# B&R Automation Studio project A2019059_Linka_Power_CP (part 14)

#### ProfinetKomunikaciaCU.st
```iecst
ACTION ProfinetKomunikaciaCU:

	//Stavy jednotky pre ovládanie kamier//
	ControlUnit.Stav_READY:= ControlUnit.Profinet_PLC_INPUTS[0].0;

END_ACTION
```

### Program Logical/Program/Linka/OvladanieSafety (IEC)

#### Main.st - Init, cyclic, exit code
```iecst
PROGRAM _INIT
	(* Insert code here *)

END_PROGRAM

PROGRAM _CYCLIC

	//*************************************Príznak tlačítka CS odblokované**********************************************//
	IF Safety.STAV.P1_Panel_TlacitkoCS_AKTIVNE AND
		Safety.STAV.P1_Robot_TlacitkoCS_AKTIVNE AND
		Safety.STAV.P1_Skrina_TlacitkoCS_AKTIVNE AND
		Safety.STAV.P2_Panel_TlacitkoCS_AKTIVNE AND
		Safety.STAV.P2_TlacitkoCS_AKTIVNE AND
		Safety.STAV.P2_Robot_TlacitkoCS_AKTIVNE AND
		Safety.STAV.P2_Skrina_TlacitkoCS_AKTIVNE AND
		Safety.STAV.P3_Skrina_TlacitkoCS_AKTIVNE AND
		Safety.STAV.P4_Panel_TlacitkoCS_AKTIVNE AND
		Safety.STAV.P4_Skrina_TlacitkoCS_AKTIVNE THEN
		Safety.STAV.TlacitkaCS_AKTIVNE:= TRUE;
	ELSE
		Safety.STAV.TlacitkaCS_AKTIVNE:= FALSE;
	END_IF

	//******************************************Reset zóny CS*******************************************************//
	IF P1_Vizu.TL_ResetCS THEN
		Safety.IN.ZonaCS_RESET:= TRUE;
		P1_Vizu.TL_ResetCS:= FALSE;
	ELSIF P2_Vizu.TL_ResetCS THEN
		Safety.IN.ZonaCS_RESET:= TRUE;
		P2_Vizu.TL_ResetCS:= FALSE;
	ELSIF P34_Vizu.TL_ResetCS THEN
		Safety.IN.ZonaCS_RESET:= TRUE;
		P34_Vizu.TL_ResetCS:= FALSE;
	END_IF

	IF Safety.IN.ZonaCS_RESET THEN
		IF Safety.STAV.ZonaCS_AKTIVNA THEN
			Safety.IN.ZonaCS_RESET:= FALSE;
		ELSIF NOT Safety.STAV.TlacitkaCS_AKTIVNE THEN
			Safety.IN.ZonaCS_RESET:= FALSE;
		END_IF
	END_IF

    //Reset bariéry vstupného výťahu//
    IF NOT Safety.STAV.P1_Vytah_Bariera_AKTIVNA THEN
        Safety.OUT.P1_ResetBarieryVytahu:= Blikac500ms;
    ELSE
        Safety.OUT.P1_ResetBarieryVytahu:= FALSE;
    END_IF

    //Reset bariéry výstupného výťahu//
    IF NOT Safety.STAV.P4_Vytah_Bariera_AKTIVNA THEN
        Safety.OUT.P4_ResetBarieryVytahu:= Blikac500ms;
    ELSE
        Safety.OUT.P4_ResetBarieryVytahu:= FALSE;
    END_IF

END_PROGRAM

PROGRAM _EXIT
	(* Insert code here *)

END_PROGRAM
```

### Program Logical/Program/Linka/OvladanieVizu (IEC)

#### Main.st - Init, cyclic, exit code
```iecst
PROGRAM _INIT
	(* Insert code here *)

END_PROGRAM

PROGRAM _CYCLIC

	//**************************************Zmena farby tlačítka Reset CS *********************************************//
	IF Safety.STAV.ZonaCS_AKTIVNA THEN
		Vizu.TL_ResetCS_Farba:= "Button_Green";
	ELSIF Safety.STAV.TlacitkaCS_AKTIVNE THEN
		IF Blikac1s THEN
			Vizu.TL_ResetCS_Farba:= "Button_Blue";
		ELSE
			Vizu.TL_ResetCS_Farba:= "Operate";
		END_IF
	ELSE
		Vizu.TL_ResetCS_Farba:= "Operate";
	END_IF

    //************************************Blokovanie tlačítok prihlásenia operátora*************************************//
    IF P1_Vizu.TL_PrihlasovOperatora_AKTIVNE THEN
        P2_Vizu.TL_PrihlasovOperatora_AKTIVNE:= FALSE;
        P34_Vizu.TL_PrihlasovOperatora_AKTIVNE:= FALSE;
        P2_Vizu.TL_PrihlasenieOperatora_ENABLE:= FALSE;
        P34_Vizu.TL_PrihlasenieOperatora_ENABLE:= FALSE;
    ELSIF P2_Vizu.TL_PrihlasovOperatora_AKTIVNE THEN
        P1_Vizu.TL_PrihlasovOperatora_AKTIVNE:= FALSE;
        P34_Vizu.TL_PrihlasovOperatora_AKTIVNE:= FALSE;
        P1_Vizu.TL_PrihlasenieOperatora_ENABLE:= FALSE;
        P34_Vizu.TL_PrihlasenieOperatora_ENABLE:= FALSE;
    ELSIF P34_Vizu.TL_PrihlasovOperatora_AKTIVNE THEN
        P1_Vizu.TL_PrihlasovOperatora_AKTIVNE:= FALSE;
        P2_Vizu.TL_PrihlasovOperatora_AKTIVNE:= FALSE;
        P1_Vizu.TL_PrihlasenieOperatora_ENABLE:= FALSE;
        P2_Vizu.TL_PrihlasenieOperatora_ENABLE:= FALSE;
    ELSE
        P1_Vizu.TL_PrihlasenieOperatora_ENABLE:= TRUE;
        P2_Vizu.TL_PrihlasenieOperatora_ENABLE:= TRUE;
        P34_Vizu.TL_PrihlasenieOperatora_ENABLE:= TRUE;
    END_IF

    //************************************Vypnutie tlačítok prihlásenie operátora*********************************************//
    //Panel 1//
    IF P1_UzivatelPrihlaseny AND P1_Vizu.TL_PrihlasovOperatora_AKTIVNE AND P1_Vizu.ActualPage <> 'PageUsers' THEN
        P1_Vizu.TL_PrihlasovOperatora_AKTIVNE:= FALSE;
    END_IF

    //Panel 2//
    IF P2_UzivatelPrihlaseny AND P2_Vizu.TL_PrihlasovOperatora_AKTIVNE THEN
        P2_Vizu.TL_PrihlasovOperatora_AKTIVNE:= FALSE;
    END_IF

    //Panel 3//
    IF P34_UzivatelPrihlaseny AND P34_Vizu.TL_PrihlasovOperatora_AKTIVNE THEN
        P34_Vizu.TL_PrihlasovOperatora_AKTIVNE:= FALSE;
    END_IF

END_PROGRAM

PROGRAM _EXIT
	(* Insert code here *)

END_PROGRAM
```

### Program Logical/Program/Pracovisko_1/P1_Main (IEC)

#### Main.st - Init, cyclic, exit code
```iecst
PROGRAM _INIT
	(* Insert code here *)

END_PROGRAM

PROGRAM _CYCLIC

	//Volanie podprogramu//
    OvlVentilovychTerminalov;
    ProfinetKomunikaciaKAM2;
    ProfinetKomunikaciaKAM3;
    ProfinetKomunikaciaKAM4;
    ProfinetKomunikaciaKAM5;
    ProfinetKomunikaciaKAM6;

    //******************************Stav moduly OK**************************************//
    IF P1_Pracovisko.STAV.ModulDI11_OK AND
        P1_Pracovisko.STAV.ModulDI12_OK AND
        P1_Pracovisko.STAV.ModulDI13_OK AND
        P1_Pracovisko.STAV.ModulDI14_OK AND
        P1_Pracovisko.STAV.ModulDM11_OK AND
        P1_Pracovisko.STAV.ModulDS11_OK AND
        P1_Pracovisko.STAV.ModulDS12_OK AND
        P1_Pracovisko.STAV.ModulSI11_OK AND
        P1_Pracovisko.STAV.ModulSI12_OK THEN
        P1_Pracovisko.STAV.Moduly_OK:= TRUE;
    ELSE
        P1_Pracovisko.STAV.Moduly_OK:= FALSE;
    END_IF

    //******************************Stav kamery OK**************************************//
    IF Linka.STAV.WenglorControlUnit_OK AND
        CAM3.STAV.READY AND
        CAM5.STAV.READY THEN
        P1_Pracovisko.STAV.Kamery_OK:= TRUE;
    ELSE
        P1_Pracovisko.STAV.Kamery_OK:= FALSE;
    END_IF

    //******************************Stav skrutkovačky OK*********************************//
    IF P1_Pracovisko.STAV.Skrutkovacka_K30_OK AND
        P1_Pracovisko.STAV.Skrutkovacka_M4_OK AND
        P1_Pracovisko.STAV.Skrutkovacka_M5_OK THEN
        P1_Pracovisko.STAV.Skrutkovacky_OK:= TRUE;
    ELSE
        P1_Pracovisko.STAV.Skrutkovacky_OK:= FALSE;
    END_IF

    //******************************Stav ventilové terminály OK***************************//
    IF P1_Pracovisko.STAV.VentilovyTerminal_VT4_OK AND P1_Pracovisko.STAV.VentilovyTerminal_VT5_OK THEN
        P1_Pracovisko.STAV.VentiloveTerminaly_OK:= TRUE;
    ELSE
        P1_Pracovisko.STAV.VentiloveTerminaly_OK:= FALSE;
    END_IF

    //Ukončenie cyklu//
    IF P1_Pracovisko.KoniecCyklu THEN
        IF P1_Vytah.Automat THEN
			P1_Vytah.KoniecCyklu:= TRUE;
		END_IF
        IF P1_Dopravniky.Automat THEN
            P1_Dopravniky.KoniecCyklu:= TRUE;
        END_IF
        IF P1_SpodnyStoper.Automat THEN
            P1_SpodnyStoper.KoniecCyklu:= TRUE;
        END_IF
        IF P1_Robot.Automat THEN
            P1_Robot.KoniecCyklu:= TRUE;
        END_IF
        IF P1_StoperSrobovania.Automat THEN
            P1_StoperSrobovania.KoniecCyklu:= TRUE;
        END_IF
        IF P1_Srobovanie.Automat THEN
            P1_Srobovanie.KoniecCyklu:= TRUE;
        END_IF
        IF P1_AkumulacnyStoper.Automat THEN
            P1_AkumulacnyStoper.KoniecCyklu:= TRUE;
        END_IF
        P1_Pracovisko.KoniecCyklu:= FALSE;
    END_IF

    //Ukončenie cyklu pri poruche//
    IF EDGEPOS(P1_PoruchaST2) THEN
        IF P1_Dopravniky.Automat THEN
            P1_Dopravniky.KoniecCyklu:= TRUE;
        END_IF
        IF P1_SpodnyStoper.Automat THEN
            P1_SpodnyStoper.KoniecCyklu:= TRUE;
        END_IF
        IF P1_Robot.Automat THEN
            P1_Robot.KoniecCyklu:= TRUE;
        END_IF
        IF P1_AkumulacnyStoper.Automat THEN
            P1_AkumulacnyStoper.KoniecCyklu:= TRUE;
        END_IF
    END_IF

    //Status prebieha ukončenie cyklu//
    IF P1_Vytah.KoniecCyklu OR
        P1_Dopravniky.KoniecCyklu OR
        P1_SpodnyStoper.KoniecCyklu OR
        P1_Robot.KoniecCyklu OR
        P1_StoperSrobovania.KoniecCyklu OR
        P1_Srobovanie.KoniecCyklu OR
        P1_AkumulacnyStoper.KoniecCyklu THEN
        P1_Pracovisko.STAV.UkoncenieCyklu_BUSY:= TRUE;
    ELSE
        P1_Pracovisko.STAV.UkoncenieCyklu_BUSY:= FALSE;
    END_IF

    //Resetovanie pracoviska po stlačení tlačítka Automat//
    IF P1_Vizu.TL_RezimAutomat THEN
        IF P1_Pracovisko.STAV.Manual THEN
            P1_Pracovisko.Reset:= TRUE;
        END_IF
        P1_Vizu.TL_RezimAutomat:= FALSE;
    END_IF

    //Resetovanie pracoviska//
    IF P1_Pracovisko.Reset THEN
        P1_Dopravniky.Reset:= TRUE;
        P1_SpodnyStoper.Reset:= TRUE;
        P1_Vytah.Reset:= TRUE;
        P1_Robot.Reset:= TRUE;
        P1_StoperSrobovania.Reset:= TRUE;
        P1_Srobovanie.Reset:= TRUE;
        P1_AkumulacnyStoper.Reset:= TRUE;
        P1_Pracovisko.Reset:= FALSE;
    END_IF

    //Prepnutie pracoviska do manualneho režimu//
    IF P1_Pracovisko.Manual THEN
        P1_Dopravniky.Manual:= TRUE;
        P1_SpodnyStoper.Manual:= TRUE;
        P1_Vytah.Manual:= TRUE;
        P1_Robot.Manual:= TRUE;
        P1_StoperSrobovania.Manual:= TRUE;
        P1_Srobovanie.Manual:= TRUE;
        P1_AkumulacnyStoper.Manual:= TRUE;
        P1_Pracovisko.Manual:= FALSE;
    END_IF

    //Spustenie pracoviska v automatickom režime//
    IF P1_Pracovisko.Automat THEN
        P1_Dopravniky.Automat:= TRUE;
        P1_SpodnyStoper.Automat:= TRUE;
        P1_Vytah.Automat:= TRUE;
        P1_Robot.Automat:= TRUE;
        P1_StoperSrobovania.Automat:= TRUE;
        P1_Srobovanie.Automat:= TRUE;
        P1_AkumulacnyStoper.Automat:= TRUE;
        P1_Pracovisko.Automat:= FALSE;
    END_IF

    //*****************************************Príznaky pracoviska******************************************//
    //Príznak pracovisko stav AUTOMAT//
    IF P1_Dopravniky.Automat OR
        P1_SpodnyStoper.Automat OR
        P1_Vytah.Automat OR
        P1_Robot.Automat OR
        P1_StoperSrobovania.Automat OR
        P1_Srobovanie.Automat OR
        P1_AkumulacnyStoper.Automat THEN
        P1_Pracovisko.STAV.Automat:= TRUE;
    ELSE
        P1_Pracovisko.STAV.Automat:= FALSE;
    END_IF

    //Priznak pracovisko stav MANUAL//
    IF P1_Dopravniky.Manual OR
        P1_SpodnyStoper.Manual OR
        P1_Vytah.Manual OR
        P1_Robot.Manual OR
        P1_StoperSrobovania.Manual OR
        P1_Srobovanie.Manual OR
        P1_AkumulacnyStoper.Manual THEN
        P1_Pracovisko.STAV.Manual:= TRUE;
    ELSE
        P1_Pracovisko.STAV.Manual:= FALSE;
    END_IF

    //Príznak pracovisko stav PoINIT//
    IF P1_Dopravniky.STAV.PoINIT AND
        P1_SpodnyStoper.STAV.PoINIT AND
        (P1_Vytah.STAV.PoINIT OR NOT P1_Vytah.Automat) AND
        P1_Robot.STAV.PoINIT AND
        P1_StoperSrobovania.STAV.PoINIT AND
        P1_Srobovanie.STAV.PoINIT AND
        P1_AkumulacnyStoper.STAV.PoINIT THEN
        P1_Pracovisko.STAV.PoINIT:= TRUE;
    ELSE
        P1_Pracovisko.STAV.PoINIT:= FALSE;
    END_IF

    //Príznak pracovisko stav READY//
    IF SC_P1_Dopravniky.Step = 1 AND
        SC_P1_SpodnyStoper.Step = 1 AND
        SC_P1_Vytah.Step = 1 AND
        SC_P1_Robot.Step = 1 AND
        SC_P1_StoperSrobovania.Step = 1 AND
        SC_P1_Srobovanie.Step = 1 AND
        SC_P1_AkumulacnyStoper.Step = 1 THEN
        P1_Pracovisko.STAV.READY:= TRUE;
    ELSE
        P1_Pracovisko.STAV.READY:= FALSE;
    END_IF

    //*****************************Zapnutie osvetlenia pracoviska*******************************************//
    IF NOT Safety.IN.P1_PredneDvere_PritomPetlice THEN
        P1_Pracovisko.OUT.OsvetlenieBunky:= TRUE;
    ELSIF NOT Safety.IN.P1_ZadneDvereLS_PritomPetlice THEN
        P1_Pracovisko.OUT.OsvetlenieBunky:= TRUE;
    ELSIF NOT Safety.IN.P1_ZadneDverePS_PritomPetlice THEN
        P1_Pracovisko.OUT.OsvetlenieBunky:= TRUE;
    ELSE
        P1_Pracovisko.OUT.OsvetlenieBunky:= FALSE;
    END_IF

    P1_Pracovisko.OUT.Osvetlenie_CAM2:= TRUE;
    P1_Pracovisko.OUT.Osvetlenie_CAM6:= TRUE;

    //****************************************Ovládanie majáka***********************************************//
    //Zelené svetlo//
    IF P1_Pracovisko.STAV.Automat THEN
        P1_Pracovisko.OUT.Majak_ZeleneSvetlo:= TRUE;
    ELSIF P1_Pracovisko.STAV.Manual THEN
        P1_Pracovisko.OUT.Majak_ZeleneSvetlo:= Blikac500ms;
    ELSE
        P1_Pracovisko.OUT.Majak_ZeleneSvetlo:= FALSE;
    END_IF

    //Žlté svetlo//
    IF P1_Pracovisko.STAV.Automat AND NOT P1_Pracovisko.STAV.PoINIT THEN
        P1_Pracovisko.OUT.Majak_ZlteSvetlo:= TRUE;
    ELSIF NOT P1_Robot.KOM_IN.Stav_RezimAUTOMAT THEN
        P1_Pracovisko.OUT.Majak_ZlteSvetlo:= Blikac500ms;
    ELSIF P1_Srobovanie.STAV.Zasobnik_K30_Prazdny THEN
        P1_Pracovisko.OUT.Majak_ZlteSvetlo:= Blikac500ms;
    ELSIF P1_Srobovanie.STAV.Zasobnik_M5_Prazdny THEN
        P1_Pracovisko.OUT.Majak_ZlteSvetlo:= Blikac500ms;
    ELSIF P1_Srobovanie.STAV.Zasobnik_M4_Prazdny THEN
        P1_Pracovisko.OUT.Majak_ZlteSvetlo:= Blikac500ms;
    ELSE
        P1_Pracovisko.OUT.Majak_ZlteSvetlo:= FALSE;
    END_IF

    //Červené svetlo//
    IF P1_Pracovisko.STAV.PORUCHA THEN
        P1_Pracovisko.OUT.Majak_CerveneSvetlo:= TRUE;
    ELSE
        P1_Pracovisko.OUT.Majak_CerveneSvetlo:= FALSE;
    END_IF

    //Zvuková signalizácia//
//    IF EDGEPOS(P1_Pracovisko.STAV.PORUCHA) THEN
//        P1_Pracovisko.OUT.Majak_Hukacka:= Blikac500ms;
//    END_IF

    IF P1_AlarmyVizu.PotvrdAlarmy THEN
        P1_Pracovisko.OUT.Majak_Hukacka:= FALSE;
    END_IF

END_PROGRAM

PROGRAM _EXIT
	(* Insert code here *)

END_PROGRAM
```

#### OvlVentilovychTerminalov.st
```iecst
ACTION OvlVentilovychTerminalov:

		//Mapovanie ventilového terminálu - VT4//
	P1_Pracovisko.OUT.VT4_OUT1.0:= P1_AkumulacnyStoper.OUT.ZasunStoper_YV74;
	P1_Pracovisko.OUT.VT4_OUT1.1:= P1_StoperSrobovania.OUT.ZasunStoper_YV110;
	P1_Pracovisko.OUT.VT4_OUT1.2:= P1_SpodnyStoper.OUT.ZasunStoper_YV111;
	P1_Pracovisko.OUT.VT4_OUT1.3:= P1_Srobovanie.OUT.ZasobSrobM4_Ofuk_RUN_YV72;
	P1_Pracovisko.OUT.VT4_OUT1.4:= P1_Srobovanie.OUT.NastrelSrobM4_NastrelSrobu_YV78;
	P1_Pracovisko.OUT.VT4_OUT1.5:= P1_Srobovanie.OUT.ZasobSrobM4_OfukTried_RUN_YV73;
	P1_Pracovisko.OUT.VT4_OUT1.6:= P1_Srobovanie.OUT.NastrelSrobM4_PosunSrobu_YV77;
	P1_Pracovisko.OUT.VT4_OUT1.7;

	P1_Pracovisko.OUT.VT4_OUT2.0:= P1_Srobovanie.OUT.SkrutkM4_PrisavSkrutky_RUN_YV81;
	P1_Pracovisko.OUT.VT4_OUT2.1:= P1_Srobovanie.OUT.SkrutkM4_OfukVakua_RUN_YV80;
	P1_Pracovisko.OUT.VT4_OUT2.2:= P1_Srobovanie.OUT.SkrutkM4_Cist_OTVOR_YV82;
	P1_Pracovisko.OUT.VT4_OUT2.3;
	P1_Pracovisko.OUT.VT4_OUT2.4:= P1_Srobovanie.OUT.SkrutkM4_Cist_POSUN_YV83;
	P1_Pracovisko.OUT.VT4_OUT2.5:= P1_Srobovanie.OUT.SkrutkM4_Cist_ODSAVANIE_YV84;
	P1_Pracovisko.OUT.VT4_OUT2.6:= P1_Srobovanie.OUT.ZasobSrobK30_Ofuk_RUN_YV85;
	P1_Pracovisko.OUT.VT4_OUT2.7:= P1_Srobovanie.OUT.ZasobSrobK30_OfukTried_RUN_YV86;

	P1_Pracovisko.OUT.VT4_OUT3.0:= P1_Srobovanie.OUT.NastrelSrobK30_PosunSrobu_YV87;
	P1_Pracovisko.OUT.VT4_OUT3.1;
	P1_Pracovisko.OUT.VT4_OUT3.2:= P1_Srobovanie.OUT.NastrelSrobK30_NastrelSrobu_YV88;
	P1_Pracovisko.OUT.VT4_OUT3.3:= P1_Srobovanie.OUT.SkrutkK30_PrisavSkrutky_RUN_YV90;
	P1_Pracovisko.OUT.VT4_OUT3.4:= P1_Srobovanie.OUT.SkrutkK30_OfukVakua_RUN_YV91;
	P1_Pracovisko.OUT.VT4_OUT3.5;
	P1_Pracovisko.OUT.VT4_OUT3.6:= P1_Srobovanie.OUT.SkrutkK30_Cist_OTVOR_YV92;
	P1_Pracovisko.OUT.VT4_OUT3.7;

	P1_Pracovisko.OUT.VT4_OUT4.0:= P1_Srobovanie.OUT.SkrutkK30_Cist_POSUN_YV123;
	P1_Pracovisko.OUT.VT4_OUT4.1:= P1_Srobovanie.OUT.SkrutkK30_Cist_ODSAVANIE_YV93;
	P1_Pracovisko.OUT.VT4_OUT4.2:= P1_Srobovanie.OUT.ZasobSrobM5_Ofuk_RUN_YV94;
	P1_Pracovisko.OUT.VT4_OUT4.3:= P1_Srobovanie.OUT.ZasobSrobM5_OfukTried_RUN_YV95;
	P1_Pracovisko.OUT.VT4_OUT4.4:= P1_Srobovanie.OUT.OddelovacSrobM5_OtocVZAD_YV102;
	P1_Pracovisko.OUT.VT4_OUT4.5:= P1_Srobovanie.OUT.OddelovacSrobM5_OtocVPRED_YV103;
	P1_Pracovisko.OUT.VT4_OUT4.6;
	P1_Pracovisko.OUT.VT4_OUT4.7;

	//Mapovanie ventilového terminálu - VT5//
	P1_Pracovisko.OUT.VT5_OUT1.0:= P1_Srobovanie.OUT.SkrutkM4_VYSUN_YV79;
	P1_Pracovisko.OUT.VT5_OUT1.1;
	P1_Pracovisko.OUT.VT5_OUT1.2:= P1_Srobovanie.OUT.SkrutkK30_VYSUN_YV89;
	P1_Pracovisko.OUT.VT5_OUT1.3;
	P1_Pracovisko.OUT.VT5_OUT1.4:= P1_Srobovanie.OUT.SkrutkM5_VYSUN_YV104;
	P1_Pracovisko.OUT.VT5_OUT1.5;
	P1_Pracovisko.OUT.VT5_OUT1.6:= P1_StoperSrobovania.OUT.VysunCentrovanie_YV112;
	P1_Pracovisko.OUT.VT5_OUT1.7:= P1_StoperSrobovania.OUT.ZasunCentrovanie_YV113;

	P1_Pracovisko.OUT.VT5_OUT2.0:= P1_Robot.OUT.OdistiGriper_YV107;
	P1_Pracovisko.OUT.VT5_OUT2.1:= P1_Robot.OUT.ZaistiGriper_YV106;
	P1_Pracovisko.OUT.VT5_OUT2.2:= P1_Robot.OUT.OtvorGriper_YV97;
	P1_Pracovisko.OUT.VT5_OUT2.3:= P1_Robot.OUT.ZatvorGriper_YV98;
	P1_Pracovisko.OUT.VT5_OUT2.4:= P1_Robot.OUT.VypniVakum_YV114;
	P1_Pracovisko.OUT.VT5_OUT2.5:= P1_Robot.OUT.ZapniVakum_YV108;
	P1_Pracovisko.OUT.VT5_OUT2.6:= P1_Srobovanie.OUT.SkrutkM5_PrisavSkrut_ZAPNI_YV105;
	P1_Pracovisko.OUT.VT5_OUT2.7:= P1_Srobovanie.OUT.SkrutkM5_PrisavSkrut_VYPNI_YV109;

	P1_Pracovisko.OUT.VT5_OUT3.0;
	P1_Pracovisko.OUT.VT5_OUT3.1;
	P1_Pracovisko.OUT.VT5_OUT3.2;
	P1_Pracovisko.OUT.VT5_OUT3.3;
	P1_Pracovisko.OUT.VT5_OUT3.4;
	P1_Pracovisko.OUT.VT5_OUT3.5;
	P1_Pracovisko.OUT.VT5_OUT3.6;
	P1_Pracovisko.OUT.VT5_OUT3.7;

	P1_Pracovisko.OUT.VT5_OUT4.0;
	P1_Pracovisko.OUT.VT5_OUT4.1;
	P1_Pracovisko.OUT.VT5_OUT4.2;
	P1_Pracovisko.OUT.VT5_OUT4.3;
	P1_Pracovisko.OUT.VT5_OUT4.4;
	P1_Pracovisko.OUT.VT5_OUT4.5;
	P1_Pracovisko.OUT.VT5_OUT4.6;
	P1_Pracovisko.OUT.VT5_OUT4.7;

END_ACTION
```

#### ProfinetKomunikaciaKAM3.st
```iecst
ACTION ProfinetKomunikaciaKAM3:

	CAM3.STAV.READY;

	//Vstupy pre kameru//
	CAM3.Profinet_PLC_OUTPUTS[0].0:= CAM3.CMD.Triger;

	//Výstupy z kamery//
	CAM3.STAV.SWITCH:= CAM3.Profinet_PLC_INPUTS[10].0;

	//Výsledky kamery//
	CAM3.RESULT.Paletka.CitanieQRkodu_DPS_OK:= CAM3.Profinet_PLC_INPUTS[0].0;

	//Prečítaný QR kód DPS//
	IF EDGE(CAM3.STAV.SWITCH) THEN
		brsstrcpy(ADR(CAM3.RESULT.Paletka.PrecitanyQRkod_DPS),ADR(CAM3.Profinet_QRkod_Znaky));
	END_IF

	//Stav výsledky READY//
	IF EDGE(CAM3.STAV.SWITCH)THEN
		CAM3.STAV.Results_READY:= TRUE;
	END_IF

	END_ACTION
```

#### ProfinetKomunikaciaKAM2.st
```iecst
ACTION ProfinetKomunikaciaKAM2:

	//Vstupy pre kameru//
	CAM2.Profinet_PLC_OUTPUTS[0].3:= CAM2.CMD.Triger;

	//Výstupy z kamery//
	CAM2.STAV.READY:= CAM2.Profinet_PLC_INPUTS[0].0;
	CAM2.STAV.SWITCH:= CAM2.Profinet_PLC_INPUTS[0].1;
    CAM2.STAV.BUSY:= CAM2.Profinet_PLC_INPUTS[0].2;
    CAM2.STAV.Command_AKCEPTOVANY:= CAM2.Profinet_PLC_INPUTS[0].3;
    CAM2.STAV.Command_READY:= CAM2.Profinet_PLC_INPUTS[0].4;
    CAM2.STAV.Command_ERROR:= CAM2.Profinet_PLC_INPUTS[0].5;

	//Výsledky kamery//
	CAM2.RESULT.Paletka.Pritom_PowerCP_5F:= CAM2.Profinet_PLC_INPUTS[2].0;
	CAM2.RESULT.Paletka.Pritom_PowerCP_4F:= CAM2.Profinet_PLC_INPUTS[2].1;
	CAM2.RESULT.Paletka.Pritom_PowerCP_5H:= CAM2.Profinet_PLC_INPUTS[2].2;
	CAM2.RESULT.Paletka.Pritom_Busbar_SpodnyLavy_5H:= CAM2.Profinet_PLC_INPUTS[2].3;
	CAM2.RESULT.Paletka.Pritom_Busbar_SpodnyPravy_5H:= CAM2.Profinet_PLC_INPUTS[2].4;
	CAM2.RESULT.Paletka.Pritom_KrytuBusbarov_5H:= CAM2.Profinet_PLC_INPUTS[2].5;
	CAM2.RESULT.Paletka.Pritom_DPS_4F5F:= CAM2.Profinet_PLC_INPUTS[2].6;
	CAM2.RESULT.Paletka.Pritom_Busbaru_Spodny_5F:= CAM2.Profinet_PLC_INPUTS[2].7;

	CAM2.RESULT.Paletka.Pritom_Busbaru_Spodny_4F:= CAM2.Profinet_PLC_INPUTS[3].0;
	CAM2.RESULT.Paletka.Pritom_Foamu_4F5F:= CAM2.Profinet_PLC_INPUTS[3].1;
	CAM2.RESULT.Paletka.Pritomn_Skeletonu_4F5F:= CAM2.Profinet_PLC_INPUTS[3].2;
	CAM2.RESULT.Paletka.Pritomn_Skeletonu_5H:= CAM2.Profinet_PLC_INPUTS[3].3;
	CAM2.RESULT.Paletka.Pritomn_LavyMVcase:= CAM2.Profinet_PLC_INPUTS[3].4;
	CAM2.RESULT.Paletka.Pritomn_PravyMVcase:= CAM2.Profinet_PLC_INPUTS[3].5;
	CAM2.RESULT.Paletka.Nepritomn_TopCoveru_4F:= CAM2.Profinet_PLC_INPUTS[3].6;
	CAM2.RESULT.Paletka.Nepritomn_TopCoveru_5F5H:= CAM2.Profinet_PLC_INPUTS[3].7;

	CAM2.RESULT.Paletka.OsadeniePlastuDPS_OK:= CAM2.Profinet_PLC_INPUTS[4].0;
	CAM2.RESULT.Paletka.KompletSpodneBusbary_OK:= CAM2.Profinet_PLC_INPUTS[4].1;

	//Stav výsledky READY//
	IF EDGE(CAM2.STAV.SWITCH)THEN
		CAM2.STAV.Results_READY:= TRUE;
	END_IF

END_ACTION
```

#### ProfinetKomunikaciaKAM4.st
```iecst
ACTION ProfinetKomunikaciaKAM4:

	//Vstupy pre kameru//
	CAM4.Profinet_PLC_OUTPUTS[0].3:= CAM4.CMD.Triger;

	//Výstupy z kamery//
	CAM4.STAV.READY:= CAM4.Profinet_PLC_INPUTS[0].0;
	CAM4.STAV.SWITCH:= CAM4.Profinet_PLC_INPUTS[0].1;
    CAM4.STAV.BUSY:= CAM4.Profinet_PLC_INPUTS[0].2;
    CAM4.STAV.Command_AKCEPTOVANY:= CAM4.Profinet_PLC_INPUTS[0].3;
    CAM4.STAV.Command_READY:= CAM4.Profinet_PLC_INPUTS[0].4;
    CAM4.STAV.Command_ERROR:= CAM4.Profinet_PLC_INPUTS[0].5;

	//Výsledky kamery//
	CAM4.RESULT.Paletka.Pritomn_Pinu1_KrytDPS_4F5F:= CAM4.Profinet_PLC_INPUTS[2].0;
	CAM4.RESULT.Paletka.Pritomn_Pinu2_KrytDPS_4F5F:= CAM4.Profinet_PLC_INPUTS[2].1;
	CAM4.RESULT.Paletka.Pritomn_Pinu3_KrytDPS_4F5F:= CAM4.Profinet_PLC_INPUTS[2].2;
	CAM4.RESULT.Paletka.Pritomn_Pinu4_KrytDPS_4F5F:= CAM4.Profinet_PLC_INPUTS[2].3;
	CAM4.RESULT.Paletka.Pritomn_Pinu5_KrytDPS_4F5F:= CAM4.Profinet_PLC_INPUTS[2].4;
	CAM4.RESULT.Paletka.Pritomn_Pinu6_KrytDPS_4F5F:= CAM4.Profinet_PLC_INPUTS[2].5;
	CAM4.RESULT.Paletka.Pritom_DPS_4F5F:= CAM4.Profinet_PLC_INPUTS[2].6;

	//Stav výsledky READY//
	IF EDGE(CAM4.STAV.SWITCH)THEN
		CAM4.STAV.Results_READY:= TRUE;
	END_IF

END_ACTION
```

#### ProfinetKomunikaciaKAM6.st
```iecst
ACTION ProfinetKomunikaciaKAM6:

	//Vstupy pre kameru//
	CAM6.Profinet_PLC_OUTPUTS[0].3:= CAM6.CMD.Triger;

	//Výstupy z kamery//
	CAM6.STAV.READY:= CAM6.Profinet_PLC_INPUTS[0].0;
	CAM6.STAV.SWITCH:= CAM6.Profinet_PLC_INPUTS[0].1;
    CAM6.STAV.BUSY:= CAM6.Profinet_PLC_INPUTS[0].2;
    CAM6.STAV.Command_AKCEPTOVANY:= CAM6.Profinet_PLC_INPUTS[0].3;
    CAM6.STAV.Command_READY:= CAM6.Profinet_PLC_INPUTS[0].4;
    CAM6.STAV.Command_ERROR:= CAM6.Profinet_PLC_INPUTS[0].5;

	//Výsledky kamery//
	CAM6.RESULT.Paletka.Pritom_SpodnychBusbarov_5H:= CAM6.Profinet_PLC_INPUTS[2].0;
	CAM6.RESULT.Paletka.Pritom_KrytuBusbarov_5H:= CAM6.Profinet_PLC_INPUTS[2].1;
	CAM6.RESULT.PowerCP.Nepritom_LavyFoam_4F5F:= CAM6.Profinet_PLC_INPUTS[2].2;
	CAM6.RESULT.PowerCP.Nepritom_PravyFoam_4F5F:= CAM6.Profinet_PLC_INPUTS[2].3;
	CAM6.RESULT.Paletka.Pritom_SpodnyBusbar_5F:= CAM6.Profinet_PLC_INPUTS[2].4;
	CAM6.RESULT.Paletka.Pritom_SpodnyBusbar_4F:= CAM6.Profinet_PLC_INPUTS[2].5;
	CAM6.RESULT.PowerCP.Pritom_LavejSkrutkyK30:= CAM6.Profinet_PLC_INPUTS[2].6;
	CAM6.RESULT.PowerCP.Pritom_PravejSkrutkyK30:= CAM6.Profinet_PLC_INPUTS[2].7;

	CAM6.RESULT.PowerCP.Pritom_SkrutkyDPS_4F5F:= CAM6.Profinet_PLC_INPUTS[3].0;
	CAM6.RESULT.PowerCP.Nepritom_ZadnejSkrutkyM4_4F:= CAM6.Profinet_PLC_INPUTS[3].1;
	CAM6.RESULT.PowerCP.Nepritom_ZadnejSkrutkyM4_5F:= CAM6.Profinet_PLC_INPUTS[3].2;
	CAM6.RESULT.PowerCP.Nepritom_PrednejSkrutkyM4_4F:= CAM6.Profinet_PLC_INPUTS[3].3;
	CAM6.RESULT.PowerCP.Nepritom_PrednejSkrutkyM4_5F:= CAM6.Profinet_PLC_INPUTS[3].4;
	CAM6.RESULT.PowerCP.Pritom_StrednejSkrutkyM5_5H:= CAM6.Profinet_PLC_INPUTS[3].5;
	CAM6.RESULT.PowerCP.Pritom_LavejSkrutkyM5_5H:= CAM6.Profinet_PLC_INPUTS[3].6;
	CAM6.RESULT.PowerCP.Pritom_PravejSkrutkyM5_5H:= CAM6.Profinet_PLC_INPUTS[3].7;

	CAM6.RESULT.Paletka.Pritom_LavyFoam_4F5F:= CAM6.Profinet_PLC_INPUTS[4].0;
	CAM6.RESULT.Paletka.Pritom_PravyFoam_4F5F:= CAM6.Profinet_PLC_INPUTS[4].1;

	//Stav výsledky READY//
	IF EDGE(CAM6.STAV.SWITCH)THEN
		CAM6.STAV.Results_READY:= TRUE;
	END_IF

END_ACTION
```

#### ProfinetKomunikaciaKAM5.st
```iecst
ACTION ProfinetKomunikaciaKAM5:

	CAM5.STAV.READY;

	//Vstupy pre kameru//
	CAM5.Profinet_PLC_OUTPUTS[0].0:= CAM5.CMD.Triger;

	//Výstupy z kamery//
	CAM5.STAV.SWITCH:= CAM5.Profinet_PLC_INPUTS[10].0;

	//Výsledky kamery//
	CAM5.RESULT.PowerCP.CitanieQRkodu_PowerCP_OK:= CAM5.Profinet_PLC_INPUTS[0].0;

	//Prečítaný QR kód DPS//
	IF EDGE(CAM5.STAV.SWITCH) THEN
		brsstrcpy(ADR(CAM5.RESULT.PowerCP.PrecitanyQRkod_PowerCP),ADR(CAM5.Profinet_QRkod_Znaky));
	END_IF

	//Stav výsledky READY//
	IF EDGE(CAM5.STAV.SWITCH)THEN
		CAM5.STAV.Results_READY:= TRUE;
	END_IF

END_ACTION
```

### Program Logical/Program/Pracovisko_1/P1_Dopravniky (IEC)

#### Main.st - Init, cyclic, exit code
```iecst
PROGRAM _INIT
	(* Insert code here *)

END_PROGRAM

PROGRAM _CYCLIC

		//Volanie funkcie SequenceControl//
	SequenceControl(SC:= SC_P1_Dopravniky);

	//Reset sekcie //
	IF NOT Safety.STAV.P1_ZonaBunky_AKTIVNA THEN
		SC_P1_Dopravniky.Step:= 0;
	ELSIF P1_Dopravniky.Reset THEN
		SC_P1_Dopravniky.Step:= 0;
		P1_Dopravniky.Reset:= FALSE;
	END_IF

	CASE SC_P1_Dopravniky.Step OF

		0:
			SC_P1_Dopravniky.StepName:='0 - Nulovanie';
			P1_Dopravniky.Automat:= FALSE;
			P1_Dopravniky.KoniecCyklu:= FALSE;
			P1_Dopravniky.Manual:= FALSE;
			P1_Dopravniky.STAV.PoINIT:= FALSE;
			P1_Dopravniky.OUT.HornyDoprav_ChodVPRED_M32:= FALSE;
			P1_Dopravniky.OUT.SpodnyDoprav_ChodVPRED_M29:= FALSE;

			IF Safety.STAV.P1_ZonaBunky_AKTIVNA AND NOT P1_Pracovisko.STAV.PORUCHA AND P1_Pracovisko.IN.PrivodVzduchu_SnimacTlaku_S18 THEN
				SC_P1_Dopravniky.ResetStep:= TRUE;
				SC_P1_Dopravniky.Step:= 1;
			END_IF

		1:
			SC_P1_Dopravniky.StepName:='1 - Cakam na spustenie vyroby';
			P1_Dopravniky.KoniecCyklu:= FALSE;
            IF P1_Dopravniky.Automat THEN
				SC_P1_Dopravniky.Step:= 2;
			ELSIF P1_Dopravniky.Manual THEN
				SC_P1_Dopravniky.Step:= 700;
			END_IF

			//********************************************************Inicializácia****************************************************************************//

		2:
			SC_P1_Dopravniky.StepName:='2 - Inicializacia - cakam na spustenie inicializacie';
			SC_P1_Dopravniky.IdleTime.PT:= T#2s;
			SC_P1_Dopravniky.AlarmTime.PT:= T#5s;

			IF P1_Srobovacky_VychodziaPozicia AND P1_Robot.STAV.PoINIT THEN
				SC_P1_Dopravniky.IdleTime.IN:= TRUE;
			ELSE
				SC_P1_Dopravniky.IdleTime.IN:= FALSE;
			END_IF

			IF SC_P1_Dopravniky.IdleTime.Q THEN
				SC_P1_Dopravniky.ResetStep:= TRUE;
				SC_P1_Dopravniky.Step:= 3;
			END_IF

		3:
			SC_P1_Dopravniky.StepName:='3 - Inicializacia - inicializacia stoprov';
			SC_P1_Dopravniky.IdleTime.PT:= T#1s;
			SC_P1_Dopravniky.AlarmTime.PT:= T#5s;

			IF NOT P1_StoperSrobovania.IN.PritomnostPaletky_S16 THEN
				P1_StoperSrobovania.OUT.ZasunStoper_YV110:= TRUE;
				SC_P1_Dopravniky.IdleTime.IN:= TRUE;
			ELSE
				SC_P1_Dopravniky.ResetStep:= TRUE;
				SC_P1_Dopravniky.Step:= 5;
			END_IF

			IF P1_StoperSrobovania.OUT.ZasunStoper_YV110 AND SC_P1_Dopravniky.IdleTime.Q THEN
				P1_StoperSrobovania.OUT.ZasunStoper_YV110:= FALSE;
				SC_P1_Dopravniky.ResetStep:= TRUE;
				SC_P1_Dopravniky.Step:= 5;
			END_IF

		5:
			SC_P2_Dopravniky.StepName:='5 - Inicializacia - ukoncenie inicializacie';
			SC_P2_Dopravniky.IdleTime.PT:= T#4s;
			SC_P2_Dopravniky.AlarmTime.PT:= T#5s;

			P1_Dopravniky.OUT.HornyDoprav_ChodVPRED_M32:= TRUE;
			P1_Dopravniky.OUT.SpodnyDoprav_ChodVPRED_M29:= TRUE;
			SC_P1_Dopravniky.IdleTime.IN:= TRUE;

			IF SC_P1_Dopravniky.IdleTime.Q THEN
				P1_Dopravniky.STAV.PoINIT:= TRUE;
				SC_P1_Dopravniky.ResetStep:= TRUE;
				SC_P1_Dopravniky.Step:= 100;
			END_IF

			//********************************************************Automatický režim****************************************************************************//

		100:
			SC_P1_Dopravniky.StepName:='100 - Automaticky Rezim - cakam na vypnutie dopravnikou';
			SC_P1_Dopravniky.IdleTime.PT:= T#200ms;
			SC_P1_Dopravniky.AlarmTime.PT:= T#5s;

			IF P1_Dopravniky.KoniecCyklu AND NOT P1_StoperSrobovania.Automat AND NOT P1_AkumulacnyStoper.Automat THEN
				SC_P1_Dopravniky.ResetStep:= TRUE;
				SC_P1_Dopravniky.Step:= 0;
			END_IF

			//*******************************************************Manuálny režim*******************************************************************************//
		700:
			SC_P1_Dopravniky.StepName:='700 - Manualny Rezim';
			SC_P1_Dopravniky.IdleTime.PT:= T#8s;
			SC_P1_Dopravniky.AlarmTime.PT:= T#5s;

	END_CASE

END_PROGRAM

PROGRAM _EXIT
	(* Insert code here *)

END_PROGRAM
```

### Program Logical/Program/Pracovisko_1/P1_SpodnyStoper (IEC)

#### Main.st - Init, cyclic, exit code
```iecst
PROGRAM _INIT
	(* Insert code here *)

END_PROGRAM

PROGRAM _CYCLIC

	//Volanie funkcie SequenceControl//
	SequenceControl(SC:= SC_P1_SpodnyStoper);

	//Reset sekcie //
	IF NOT Safety.STAV.P1_ZonaBunky_AKTIVNA THEN
		SC_P1_SpodnyStoper.Step:= 0;
	ELSIF P1_SpodnyStoper.Reset THEN
		SC_P1_SpodnyStoper.Step:= 0;
		P1_SpodnyStoper.Reset:= FALSE;
	END_IF

	CASE SC_P1_SpodnyStoper.Step OF

		0:
			SC_P1_SpodnyStoper.StepName:='0 - Nulovanie';
			P1_SpodnyStoper.Automat:= FALSE;
			P1_SpodnyStoper.KoniecCyklu:= FALSE;
			P1_SpodnyStoper.Manual:= FALSE;
			P1_SpodnyStoper.STAV.PoINIT:= FALSE;
			P1_SpodnyStoper.OUT.ZasunStoper_YV111:= FALSE;

			IF Safety.STAV.P1_ZonaBunky_AKTIVNA AND NOT P1_Pracovisko.STAV.PORUCHA AND P1_Pracovisko.IN.PrivodVzduchu_SnimacTlaku_S18 THEN
				SC_P1_SpodnyStoper.ResetStep:= TRUE;
				SC_P1_SpodnyStoper.Step:= 1;
			END_IF

		1:
			SC_P1_SpodnyStoper.StepName:='1 - Cakam na spustenie vyroby';
			P1_SpodnyStoper.KoniecCyklu:= FALSE;
            IF P1_SpodnyStoper.Automat THEN
				SC_P1_SpodnyStoper.Step:= 2;
			ELSIF P1_SpodnyStoper.Manual THEN
				SC_P1_SpodnyStoper.Step:= 700;
			END_IF

			//********************************************************Inicializácia****************************************************************************//
		2:
			SC_P1_SpodnyStoper.StepName:='2 - Inicializacia - cakam na spustenie inicializacie';
			SC_P1_SpodnyStoper.IdleTime.PT:= T#4s;
			SC_P1_SpodnyStoper.AlarmTime.PT:= T#5s;

			IF P1_Dopravniky.STAV.PoINIT THEN
				SC_P1_SpodnyStoper.ResetStep:= TRUE;
				SC_P1_SpodnyStoper.Step:= 3;
			END_IF

		3:
			SC_P1_SpodnyStoper.StepName:='3 - Inicializacia - hladanie paletky';
			SC_P1_SpodnyStoper.IdleTime.PT:= T#5s;
			SC_P1_SpodnyStoper.AlarmTime.PT:= T#5s;
			SC_P1_SpodnyStoper.IdleTime.IN:= TRUE;

			IF P1_SpodnyStoper.IN.PritomnPaletky_IS64 THEN
				P1_SpodnyStoper.STAV.PoINIT:= TRUE;
				SC_P1_SpodnyStoper.ResetStep:= TRUE;
				SC_P1_SpodnyStoper.Step:= 101;
			ELSIF SC_P1_SpodnyStoper.IdleTime.Q THEN
				P1_SpodnyStoper.STAV.PoINIT:= TRUE;
				SC_P1_SpodnyStoper.ResetStep:= TRUE;
				SC_P1_SpodnyStoper.Step:= 100;
			END_IF

			//********************************************************Automatický režim****************************************************************************//
		100:
			SC_P1_SpodnyStoper.StepName:='100 - Automaticky Rezim - cakam na príchod paletky na stoper';
			SC_P1_SpodnyStoper.IdleTime.PT:= T#200ms;
			SC_P1_SpodnyStoper.AlarmTime.PT:= T#5s;

			SC_P1_SpodnyStoper.IdleTime.IN:= P1_SpodnyStoper.IN.PritomnPaletky_IS64;

            IF P1_SpodnyStoper.KoniecCyklu THEN
                SC_P1_SpodnyStoper.ResetStep:= TRUE;
                SC_P1_SpodnyStoper.Step:= 0;
            ELSIF SC_P1_SpodnyStoper.IdleTime.Q THEN
				SC_P1_SpodnyStoper.ResetStep:= TRUE;
				SC_P1_SpodnyStoper.Step:= 101;
			END_IF

		101:
			SC_P1_SpodnyStoper.StepName:='101 - Automaticky Rezim - cakam na vyvezenie paletky na dopravnik vytahu';
			SC_P1_SpodnyStoper.IdleTime.PT:= T#200ms;
			SC_P1_SpodnyStoper.AlarmTime.PT:= T#5s;

            IF P1_SpodnyStoper.KoniecCyklu THEN
                SC_P1_SpodnyStoper.ResetStep:= TRUE;
                SC_P1_SpodnyStoper.Step:= 0;
            ELSIF SC_P1_Vytah.Step = 105 AND NOT P1_Vytah.IN.PritomnostPaletky_S19 THEN
				SC_P1_SpodnyStoper.ResetStep:= TRUE;
				SC_P1_SpodnyStoper.Step:= 105;
			ELSIF NOT P1_SpodnyStoper.IN.PritomnPaletky_IS64 THEN
				SC_P1_SpodnyStoper.ResetStep:= TRUE;
				SC_P1_SpodnyStoper.Step:= 100;
			END_IF

		105:
			SC_P1_SpodnyStoper.StepName:='105 - Automaticky Rezim - vyvazam paletku na dopravnik vytahu';
			SC_P1_SpodnyStoper.IdleTime.PT:= T#200ms;
			SC_P1_SpodnyStoper.AlarmTime.PT:= T#10s;

			IF NOT SC_P1_SpodnyStoper.Switch1 THEN
				P1_SpodnyStoper.OUT.ZasunStoper_YV111:= TRUE;
				SC_P1_SpodnyStoper.AlarmTime.IN:= TRUE;
                SC_P1_SpodnyStoper.Switch1:= TRUE;
			END_IF

			IF NOT P1_SpodnyStoper.IN.PritomnPaletky_IS64 THEN
                P1_SpodnyStoper.OUT.ZasunStoper_YV111:= FALSE;
                SC_P1_SpodnyStoper.AlarmTime.IN:= FALSE;
			END_IF

			IF P1_Vytah.IN.PritomnostPaletky_S19 AND NOT P1_SpodnyStoper.OUT.ZasunStoper_YV111 THEN
				SC_P1_SpodnyStoper.ResetStep:= TRUE;
				SC_P1_SpodnyStoper.Step:= 100;
			END_IF

            IF SC_P1_SpodnyStoper.AlarmTime.Q THEN
                P1_Alarmy[163]:= TRUE;
                P1_Pracovisko.KoniecCyklu:= TRUE;
                SC_P1_SpodnyStoper.ResetStep:= TRUE;
                SC_P1_SpodnyStoper.Step:= 0;
            END_IF

			//*******************************************************Manuálny režim*******************************************************************************//
		700:
			SC_P1_SpodnyStoper.StepName:='700 - Manualny Rezim';
			SC_P1_SpodnyStoper.IdleTime.PT:= T#8s;
			SC_P1_SpodnyStoper.AlarmTime.PT:= T#5s;

	END_CASE

			END_PROGRAM

PROGRAM _EXIT
			(* Insert code here *)

			END_PROGRAM
```

### Program Logical/Program/Pracovisko_1/P1_StoperSrobovania (IEC)
